INTERFACE I_TimeSpanConversions

// Converts the time span represented by the instance into days.
METHOD ToDays : ULINT // The total number of days in the time span.
VAR_INPUT
END_VAR
END_METHOD

// Converts the time span represented by the instance into hours.
METHOD ToHours : ULINT // The total number of hours in the time span.
VAR_INPUT
END_VAR
END_METHOD

// Converts the time span represented by the instance into microseconds.
METHOD ToMicroseconds : ULINT // The total number of microseconds in the time span.
VAR_INPUT
END_VAR
END_METHOD

// Converts the time span represented by the instance into milliseconds.
METHOD ToMilliseconds : ULINT // The total number of milliseconds in the time span.
VAR_INPUT
END_VAR
END_METHOD

// Converts the time span represented by the instance into minutes.
METHOD ToMinutes : ULINT // The total number of minutes in the time span.
VAR_INPUT
END_VAR
END_METHOD

// Converts the time span represented by the instance into nanoseconds.
METHOD ToNanoseconds : ULINT // The total number of nanoseconds in the time span.
VAR_INPUT
END_VAR
END_METHOD

// Converts the time span represented by the instance into seconds.
METHOD ToSeconds : ULINT // The total number of seconds in the time span.
VAR_INPUT
END_VAR
END_METHOD

END_INTERFACE

(* stored: Version 1.1.0.1
   Itf I_TimeSpanConversions: Id {c9e0566c-f7f4-0284-1189-fb285bffe885}
   Method ToDays: Id {5c75e9c3-e8af-0940-1aa8-b7930e311c22}
   Method ToHours: Id {e1f7ea57-493e-0784-1ed0-8bdee7448705}
   Method ToMicroseconds: Id {a469b6d9-f20a-0fbd-1991-ffff26eaae98}
   Method ToMilliseconds: Id {247c5852-f991-082d-2538-f01d0ece2aa0}
   Method ToMinutes: Id {4aee05cc-6553-0562-01fb-ec6c2d389694}
   Method ToNanoseconds: Id {ab38f017-7796-02d4-1089-090badd0b56c}
   Method ToSeconds: Id {670de2a8-88b0-0762-32ca-ebede3078c65} *)
